{attribute addProperty BoxType "AMP8000-0030-0103-0103"}
{attribute addProperty Id "FSOEAT %I*FSOE_83CE5B3E81"}
{attribute addProperty CRC "367935978"}
{attribute addProperty SizeInBites "8"}
{attribute addProperty SizeInBytes "1"}
TYPE Standard_Inputdata_15EE41EA :
STRUCT
	{attribute addProperty Name "FSOE"}
	FSOE AT %I* : FSOE_83CE5B3E;
END_STRUCT
END_TYPE

(* stored: Version 1.2.0.0, ProductVersion 3.1.4024.9
   DUT Standard_Inputdata_15EE41EA: Id {7d4c3f48-015f-4e8f-8272-56def55624e0} *)
